(* IEC 61131-3 sources: MotionProf/, 9 files *)

(* ---- MotionProf.typ ---- *)
TYPE
	MotionProfMoveEnum :
		( (*Movement types*)
		MOTIONPROF_MOVE_NONE := 0, (*Undefined profile*)
		MOTIONPROF_MOVE_ZERO := 1, (*Zero acceleration profile*)
		MOTIONPROF_MOVE_DEC := 2, (*Decelerate then accelerate profile*)
		MOTIONPROF_MOVE_ACC := 3, (*Decelerate then accelerate profile*)
		MOTIONPROF_MOVE_DECACC := 10, (*Decelerate then accelerate profile*)
		MOTIONPROF_MOVE_DECACC_SATURATED := 11, (*Decelerate, saturate at min velocity, accelerate profile*)
		MOTIONPROF_MOVE_ACCDEC := 12, (*Accelerate then decelerate profile*)
		MOTIONPROF_MOVE_ACCDEC_SATURATED := 13, (*Accelerate, saturate at max velocity, decelerate profile*)
		MOTIONPROF_MOVE_DECDEC := 20, (*Decelerate, hold at intermediate velocity, decelerate profile*)
		MOTIONPROF_MOVE_ACCACC := 21 (*Accelerate, hold at intermediate velocity, accelerate profile*)
		);
	MotionProfProfileType : 	STRUCT  (*Profile structure*)
		NumberOfPoints : USINT; (*Number of points in profile*)
		TimePoints : ARRAY[0..4]OF LREAL; (*[s] Time points*)
		Distance : LREAL; (*[units] Distance*)
		VelocityPoints : ARRAY[0..4]OF LREAL; (*[units/s] Velocity points*)
		Acceleration : LREAL; (*[units/s/s] Acceleration magnitude*)
		MoveType : MotionProfMoveEnum; (*Movement type*)
	END_STRUCT;
	MotionProfBaseOutputType : 	STRUCT  (*Base output structure*)
		t_ : ARRAY[0..3]OF LREAL; (*[s] Time points*)
		dx : LREAL; (*[units] Distance*)
		v_ : ARRAY[0..3]OF LREAL; (*[units/s] Velocity points*)
		a : LREAL; (*[units/s/s] Acceleration magnitude*)
		move : MotionProfMoveEnum; (*Movement type*)
	END_STRUCT;
	MotionProfPointOutputType : 	STRUCT  (*Time series point output structure*)
		x : LREAL; (*[units] Position*)
		v : LREAL; (*[units/s] Velocity*)
		a : LREAL; (*[units/s/s] Acceleration*)
		j : LREAL; (*[units/s/s/s] Jerk*)
	END_STRUCT;
	MotionProfTimeDiffOutputType : 	STRUCT  (*Time duration difference output structure*)
		dt_tilde : LREAL; (*Difference in time durations*)
		AccDec : MotionProfBaseOutputType; (*AccDec profile*)
		DecAcc : MotionProfBaseOutputType; (*DecAcc profile*)
	END_STRUCT;
END_TYPE

(* ---- PathPlan.typ ---- *)
TYPE
	PathPlanMoveEnum :
		( (*Profile movement type*)
		PATH_MOVE_NONE := 0, (*Undefined movement*)
		PATH_MOVE_DECACCPEAK := 1, (*Profile decelerates then accelerates*)
		PATH_MOVE_DECACCSATURATED := 2, (*Profile decelerates, saturates, then accelerates*)
		PATH_MOVE_ACCDECPEAK := 10, (*Profile accelerates then decelerates*)
		PATH_MOVE_ACCDECSATURATED := 20, (*Profile accelerates, saturates, then decelerates*)
		PATH_MOVE_DECDEC := 30, (*Profile decelerates, holds velocity, then decelerates*)
		PATH_MOVE_ACCACC := 40 (*Profile accelerates, holds velocity, then accelerates*)
		);
	PathPlanErrorEnum :
		( (*Return code for all functions*)
		PATH_ERROR_NONE := 0, (*Successful completion*)
		PATH_ERROR_VELOCITYLIMIT := 10, (*Implausible velocity limits*)
		PATH_ERROR_VELOCITYENDPT := 11, (*Velocity endpoints exceed limits*)
		PATH_ERROR_NONPOSITIVE := 12, (*Non-positive time, distance, or acceleration input*)
		PATH_ERROR_MOVELIMIT := 13, (*Input values require impossible or infinite acceleration magnitude*)
		PATH_ERROR_NOSOLUTION2ND := 20, (*2nd order polynomial has imaginary roots*)
		PATH_ERROR_NOSOLUTION1ST := 21, (*1st order polynomianl has no roots*)
		PATH_ERROR_POINTLIMIT := 30, (*Number of points exceeds range [2, PATH_POINTS_INDEX + 1]*)
		PATH_ERROR_TIMESEQUENCE := 31, (*Time points are not sequential*)
		PATH_ERROR_TIMELIMIT := 32, (*Request time exceeds time points*)
		PATH_ERROR_JERKLIMIT := 33 (*Jerk factor exceeds range [1.0, 2.0]*)
		);
	PathPlanBaseSolutionType : 	STRUCT  (*Solution structure for base functions*)
		t_ : ARRAY[0..3]OF LREAL; (*[s] Time points, t_[0] always 0.0*)
		dx : LREAL; (*[Units] Distance*)
		v_ : ARRAY[0..3]OF LREAL; (*[Units/s] Velocity points, v_[0] = v_0 and v_[3] = v_f*)
		a : LREAL; (*[Units/s^2] Acceleration magnitude*)
		move : PathPlanMoveEnum; (*Movement type*)
	END_STRUCT;
	PathPlanRootsSolutionType : 	STRUCT  (*2nd order (quadratic) roots solution *)
		r_1 : LREAL; (*First real root*)
		r_2 : LREAL; (*Second real root*)
	END_STRUCT;
	PathPlanInTimeSolutionType : 	STRUCT  (*Solution structure for time difference functions*)
		accDec : PathPlanInTimePathType; (*Acc/Dec profile*)
		decAcc : PathPlanInTimePathType; (*Dec/Acc profile*)
		dt_tilde : LREAL; (*[s] Difference in time durations*)
	END_STRUCT;
	PathPlanInTimePathType : 	STRUCT  (*Path structure for time difference functions*)
		t_ : ARRAY[0..4]OF LREAL; (*[s] Time points*)
		dx : LREAL; (*[Units] Distance*)
		v_ : ARRAY[0..4]OF LREAL; (*[Units/s] Velocity points*)
		a : LREAL; (*[Units/s^2] Acceleration magnitude*)
		move : PathPlanMoveEnum; (*Move type*)
	END_STRUCT;
	PathPlanPointSolutionType : 	STRUCT  (*Interpolated point solution of linear segments with parabolic blends*)
		x : LREAL; (*[Units] Position*)
		v : LREAL; (*[Units/s] Velocity*)
		a : LREAL; (*[Units/s^2] Acceleration*)
		j : LREAL; (*[Units/s^3] Jerk*)
	END_STRUCT;
END_TYPE

(* ---- Types.typ ---- *)
TYPE
	PathPlanMoveEnum :
		(
		PATH_MOVE_NONE := 0,
		PATH_DEC_ACC_PEAK := 1,
		PATH_DEC_ACC_SATURATED := 2,
		PATH_ACC_DEC_PEAK := 10,
		PATH_ACC_DEC_SATURATED := 20,
		PATH_DEC_DEC := 30,
		PATH_ACC_ACC := 40
		);
	PathPlanErrorCode :
		( (*Return code for all functions*)
		PATH_ERROR_NONE, (*No error has occured*)
		PATH_ERROR_TIME_LIMIT, (*The time duration exceeds possible limits given input values*)
		PATH_ERROR_DIST_LIMIT, (*The distance exceeds possible limits given input values*)
		PATH_ERROR_VEL_LIMITS_INVALID, (*Invalid velocity limits*)
		PATH_ERROR_VEL_ENDPT_LIMIT, (*The velocity endpoint(s) exceeds the specified velocity limits*)
		PATH_ERROR_ACC_LIMIT, (*The given input parameters would require an infinite acceleration to complete the move*)
		PATH_ERROR_NONPOS_INPUT, (*Time duration, distance, and/or acceleration input value is non-positive*)
		PATH_ERROR_HIGHER_ORDER,
		PATH_ERROR_2ND_ORDER_NO_SOLN, (*The 2nd order equation's solution results in imaginary roots*)
		PATH_ERROR_1ST_ORDER_NO_SOLN, (*The 1st order equation has no solution (constant)*)
		PATH_ERROR_POINT_LIMIT,
		PATH_ERROR_SEQ_POINTS,
		PATH_ERROR_TIME_POINT (*The requested time value exceeds the provided velocity profile*)
		);
	PathPlanBaseSolutionType : 	STRUCT
		t : ARRAY[0..3]OF REAL;
		dx : REAL;
		v : ARRAY[0..3]OF REAL;
		a : REAL;
		Move : PathPlanMoveEnum;
	END_STRUCT;
	PathPlanTimeDiffSolutionType : 	STRUCT
		tA : ARRAY[0..3]OF REAL;
		vA : ARRAY[0..3]OF REAL;
		MoveA : PathPlanMoveEnum;
		tB : ARRAY[0..3]OF REAL;
		vB : ARRAY[0..3]OF REAL;
		MoveB : PathPlanMoveEnum;
		tdiff : REAL;
		a : REAL;
	END_STRUCT;
	PathPlanPointSolutionType : 	STRUCT
		x : REAL;
		v : REAL;
		a : REAL;
	END_STRUCT;
END_TYPE

(* ---- MotionProf.fun ---- *)
FUNCTION MotionProfAcc : DINT (*Minimum acceleration to move in time over a distance*)
	VAR_INPUT
		Duration : LREAL; (*[s] Time duration*)
		Distance : LREAL; (*[units] Distance*)
		InitialVelocity : LREAL; (*[units/s] Initial velocity*)
		FinalVelocity : LREAL; (*[units/s] Final velocity*)
		MinimumVelocity : LREAL; (*[units/s] Minimum velocity*)
		MaximumVelocity : LREAL; (*[units/s] Maximum velocity*)
	END_VAR
	VAR_IN_OUT
		Profile : MotionProfProfileType; (*Profile output*)
	END_VAR
END_FUNCTION

FUNCTION MotionProfTime : DINT (*Minimum time duration to move with acceleration over a distance*)
	VAR_INPUT
		Distance : LREAL; (*[units] Distance*)
		InitialVelocity : LREAL; (*[units/s] Initial velocity*)
		FinalVelocity : LREAL; (*[units/s] Final velocity*)
		MinimumVelocity : LREAL; (*[units/s] Minimum velocity*)
		MaximumVelocity : LREAL; (*[units/s] Maximum velocity*)
		Acceleration : LREAL; (*[units/s/s] Acceleration magnitude*)
	END_VAR
	VAR_IN_OUT
		Profile : MotionProfProfileType; (*Profile output*)
	END_VAR
END_FUNCTION

FUNCTION MotionProfDist : DINT (*Maximum distance from move with acceleration in time*)
	VAR_INPUT
		Duration : LREAL; (*[s] Time duration*)
		InitialVelocity : LREAL; (*[units/s] Initial velocity*)
		FinalVelocity : LREAL; (*[units/s] Final velocity*)
		MinimumVelocity : LREAL; (*[units/s] Minimum velocity*)
		MaximumVelocity : LREAL; (*[units/s] Maximum velocity*)
		Acceleration : LREAL; (*[units/s/s] Acceleration magnitude*)
	END_VAR
	VAR_IN_OUT
		Profile : MotionProfProfileType; (*Profile output*)
	END_VAR
END_FUNCTION

FUNCTION MotionProfVel : DINT (*Minimum velocity to move with acceleration in time over a distance*)
	VAR_INPUT
		Duration : LREAL; (*[s] Time duration*)
		Distance : LREAL; (*[units] Distance*)
		InitialVelocity : LREAL; (*[units/s] Initial velocity*)
		FinalVelocity : LREAL; (*[units/s] Final velocity*)
		MinimumVelocity : LREAL; (*[units/s] Minimum velocity*)
		MaximumVelocity : LREAL; (*[units/s] Maximum velocity*)
		Acceleration : LREAL; (*[units/s/s] Acceleration magnitude*)
	END_VAR
	VAR_IN_OUT
		Profile : MotionProfProfileType; (*Profile output*)
	END_VAR
END_FUNCTION

FUNCTION MotionProfTimeDiff : DINT (*Maximum difference in time duration between fastest and slowest profiles*)
	VAR_INPUT
		Distance : LREAL; (*[units] Distance*)
		InitialVelocity : LREAL; (*[units/s] Initial velocity*)
		FinalVelocity : LREAL; (*[units/s] Final velocity*)
		MinimumVelocity : LREAL; (*[units/s] Minimum velocity*)
		MaximumVelocity : LREAL; (*[units/s] Maximum velocity*)
		Acceleration : LREAL; (*[units/s/s] Acceleration magnitude*)
	END_VAR
	VAR_IN_OUT
		Output : MotionProfTimeDiffType; (*Output*)
	END_VAR
END_FUNCTION

FUNCTION MotionProfAccTimeDiff : DINT (*Minimum acceleration to achieve moves throughout a time difference*)
	VAR_INPUT
		TimeDifference : LREAL; (*[s] Difference in time durations*)
		Distance : LREAL; (*[units] Distance*)
		InitialVelocity : LREAL; (*[units/s] Initial velocity*)
		FinalVelocity : LREAL; (*[units/s] Final velocity*)
		MinimumVelocity : LREAL; (*[units/s] Minimum velocity*)
		MaximumVelocity : LREAL; (*[units/s] Maximum velocity*)
	END_VAR
	VAR_IN_OUT
		Output : MotionProfTimeDiffType; (*Output*)
	END_VAR
END_FUNCTION

FUNCTION MotionProfAccTimeDiffZero : DINT (*Minimum acceleration to achieve moves throughout a time difference starting at standstill*)
	VAR_INPUT
		TimeDifference : LREAL; (*[s] Difference in time durations*)
		Distance : LREAL; (*[units] Distance*)
		FirstVelocity : LREAL; (*[units/s] First velocity point from standstill*)
		FinalVelocity : LREAL; (*[units/s] Final velocity*)
		MinimumVelocity : LREAL; (*[units/s] Minimum velocity*)
		MaximumVelocity : LREAL; (*[units/s] Maximum velocity*)
	END_VAR
	VAR_IN_OUT
		Output : MotionProfTimeDiffType; (*Output*)
	END_VAR
END_FUNCTION

FUNCTION MotionProfPoint : DINT (*Velocity profile point interpolation*)
	VAR_INPUT
		InitialPosition : LREAL; (*[units] Initial position*)
		TimePoints : ARRAY[0..MOTIONPROF_POINT_MAX] OF LREAL; (*[s] Time points*)
		VelocityPoints : ARRAY[0..MOTIONPROF_POINT_MAX] OF LREAL; (*[units/s] Velocity points*)
		NumberOfPoints : USINT; (*Number of points*)
		Time : LREAL; (*[s] Time interpolation*)
		JerkFactor : LREAL; (*Jerk factor 1.0 infinite jerk 2.0 minimum jerk*)
	END_VAR
	VAR_IN_OUT
		Point : MotionProfPointType; (*Point output*)
	END_VAR
END_FUNCTION

(* ---- PathKin.fun ---- *)
FUNCTION Kin_GetAcc : USINT
	VAR_INPUT
		dt : REAL;
		dx : REAL;
		v0 : REAL;
		vf : REAL;
		vmin : REAL;
		vmax : REAL;
	END_VAR
	VAR_IN_OUT
		soln : KinGetAccSoln_typ;
	END_VAR
END_FUNCTION

FUNCTION Kin_GetAccInTimespanPlus : USINT
	VAR_INPUT
		tdiff : REAL;
		dx : REAL;
		v1 : REAL;
		vf : REAL;
		vmin : REAL;
		vmax : REAL;
	END_VAR
	VAR_IN_OUT
		soln : KinGetAccInTimespanSoln_typ;
	END_VAR
END_FUNCTION

FUNCTION Kin_GetTimespan : USINT
	VAR_INPUT
		dx : REAL;
		v0 : REAL;
		vf : REAL;
		vmin : REAL;
		vmax : REAL;
		a : REAL;
	END_VAR
	VAR_IN_OUT
		soln : KinGetTimespanSoln_typ;
	END_VAR
END_FUNCTION

FUNCTION Kin_GetVelProfPoint : USINT
	VAR_INPUT
		x0 : REAL;
		timePoints : ARRAY[0..KIN_MAX_PROF_POINTS] OF REAL;
		velPoints : ARRAY[0..KIN_MAX_PROF_POINTS] OF REAL;
		n : USINT;
		t : REAL;
	END_VAR
	VAR_IN_OUT
		soln : KinGetVelProfPointSoln_typ;
	END_VAR
END_FUNCTION

(* ---- PathPlan.fun ---- *)
FUNCTION PathPlanAcc : DINT (*Minimum acceleration to move in time over a distance*)
	VAR_INPUT
		dt : LREAL; (*[s] Time duration*)
		dx : LREAL; (*[units] Distance*)
		v_0 : LREAL; (*[units/s] Initial velocity*)
		v_f : LREAL; (*[units/s] Final velocity*)
		v_min : LREAL; (*[units/s] Minimum velocity*)
		v_max : LREAL; (*[units/s] Maximum velocity*)
	END_VAR
	VAR_IN_OUT
		output : PathPlanBaseOutputType; (*Output*)
	END_VAR
END_FUNCTION

FUNCTION PathPlanRoots : DINT (*Find real roots of second order polynomial (quadratic equation)*)
	VAR_INPUT
		p_2 : LREAL; (*2nd order coefficient*)
		p_1 : LREAL; (*1st order coefficient*)
		p_0 : LREAL; (*0th order coefficient*)
	END_VAR
	VAR_IN_OUT
		output : PathPlanRootsOutputType; (*Output*)
	END_VAR
END_FUNCTION

(* ---- Constants.var ---- *)
VAR CONSTANT
	PATH_POINTS_MAX_INDEX : USINT := 19;
END_VAR

(* ---- MotionProf.var ---- *)
VAR CONSTANT
	MOTIONPROF_ERROR_NULL_POINTER : DINT := -5; (*Invalid point to output structure*)
	MOTIONPROF_ERROR_INPUT_VELOCITY : DINT := -1; (*Invalid input velocity limits or endpoints*)
	MOTIONPROF_ERROR_INPUT_MOVE : DINT := -2; (*The input distance or acceleration is impossible given the velocity limits*)
	MOTIONPROF_ERROR_INPUT_POSITIVE : DINT := -3; (*Input(s) are non-positive*)
	MOTIONPROF_ERROR_NO_SOLUTION : DINT := -4; (*No plausible motion profile could be found*)
	MOTIONPROF_POINT_MAX : USINT := 20; (*Maximum points in a velocity profile*)
	MOTIONPROF_PROFILE_MAX : USINT := 5; (*Maximum points in a profile*)
END_VAR

(* ---- PathPlan.var ---- *)
(*********************************************************************************
 * File: PathPlan.var
 * Author: Tyler Matijevich
 * Created: 2020-04-06
 *********************************************************************************)
VAR CONSTANT
	PATH_POINT_INDEX : USINT := 19; (*Max index of velocity-time point arrays*)
END_VAR
